TYPE PTOstatusChannel :
STRUCT
	{attribute addProperty Name "Status"}
	Status AT %I*: stPTOstatus;
END_STRUCT
END_TYPE

(* stored: Version 1.1.0.1, ProductVersion 3.1.4024.9
   DUT PTOstatusChannel: Id {dfedf5aa-6f19-09e9-09c5-74f2cbccaee3} *)
